TYPE Ch : STRING(1); END_TYPE

(* stored: Version 1.1.0.1
   DUT Ch: Id {b71b32e5-3895-434d-8583-ea43f14b4247} *)
